INTERFACE I_HostSynchronousRpcHandlers

METHOD PUBLIC RegisterHandler
VAR_INPUT
	MethodName : T_MAXSTRING;
	Handler : I_SynchronousRpcHandler;
END_VAR
END_METHOD

END_INTERFACE

(* stored: Version 1.1.0.1, ProductVersion 3.1.4024.12
   Itf I_HostSynchronousRpcHandlers: Id {da8e4899-7ba5-4826-aeb9-b187eb45a5cc}
   Method RegisterHandler: Id {24dec3f3-3d25-42e6-a499-e48d424a6e95} *)
